TYPE ST_GetBox :
STRUCT
	Info 			: ARRAY[0..200] OF ST_GetBoxInfo;
	//盒數
	NeedBox			:INT;
	//資料交握確認
	HandShake		: st_HandshakeBase;
END_STRUCT
END_TYPE

(* stored: Version 1.1.0.1, ProductVersion 3.1.4024.13
   DUT ST_GetBox: Id {fe3de813-8bf4-4153-9084-1e8e9a7b1e16} *)
